// TIA Portal V19 export
TYPE "LAF_typeDriveDiagConfig"
TITLE = LAF_typeDriveDiagConfig
// Technology Object and Sinamics configuration structure for drive diagnostic. Structure is designed to use for an array.
// stored: Access Published
   STRUCT
      referenceDesignator : WString[128];   // Name or reference designator of the drive object that is shown in HMI (value is assigned in startup OB; if value is default value, than HMI shows name of TO; if no TO is used, than HMI schows an empty string)
      axisDB : DB_ANY;   // DB number of technology object (value is assigned in startup OB; if no TO is used, axisDB = 0)
      sinaType : UInt;   // 0=NO_TYPE, 114=G120, 124=S120, 125=S120_EPOS, 220=S200, 221=S200_EPOS, 222=S210, 223=S210_EPOS
      sinaHwID : HW_IO;   // Identification of PROFINET IO device or DP slave for the Sinamics drive object (value is assigned in startup OB)
      sinaDriveObjectNo : USInt := 1;   // Sinamics drive object number (value is assigned in startup OB; if drive is single-axis, drive object numer = 1)
   END_STRUCT;
END_TYPE
